// Interface for a set implemented using a binary search tree.
INTERFACE I_Tree_Set EXTENDS I_Set

// Traversal method for retrieving values in the tree set.
PROPERTY _Traversal : T_BST_Traversal
GET
END_GET
SET
END_SET
END_PROPERTY

END_INTERFACE

(* stored: Version 1.1.0.1
   Itf I_Tree_Set: Id {cfffa3b6-c0bb-0ecd-3db9-4d890602e0ac}
   Property _Traversal: Id {1640ea1e-fc47-0b52-28be-74b61525dc0e}
   Get Get: Id {5cde1be4-6dfe-00f5-07bf-dfe1a63a9c6d}
   Set Set: Id {cce2cf53-5d42-09cf-0c8e-16b06c8dc5b8} *)
